// TIA Portal V20 export
FUNCTION "PreProcess_Safety" : Void   // FC1, LAD
{ S7_Optimized_Access := 'TRUE' }
// stored: SetENOAutomatically false
BEGIN

REGION Network 1
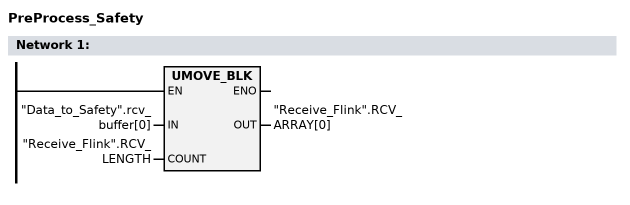
   UMOVE_BLK(IN := "Data_to_Safety".rcv_buffer[0],
             COUNT := "Receive_Flink".RCV_LENGTH,
             OUT => "Receive_Flink".RCV_ARRAY[0]);
END_REGION
END_FUNCTION
